Fanuc TP program (LS listing): SET_STR.LS

/PROG  SET_STR
/ATTR
OWNER		= MNEDITOR;
COMMENT		= "";
PROG_SIZE	= 228;
CREATE		= DATE 26-06-16  TIME 17:54:20;
MODIFIED	= DATE 26-06-16  TIME 17:54:20;
FILE_NAME	= SET_STR;
VERSION		= 0;
LINE_COUNT	= 2;
MEMORY_SIZE	= 592;
PROTECT		= READ_WRITE;
TCD:  STACK_SIZE	= 0,
      TASK_PRIORITY	= 50,
      TIME_SLICE	= 0,
      BUSY_LAMP_OFF	= 0,
      ABORT_REQUEST	= 0,
      PAUSE_REQUEST	= 0;
DEFAULT_GROUP	= 1,*,*,*,*;
CONTROL_CODE	= 00000000 00000000;
LOCAL_REGISTERS	= 0,0,0;
/APPL
/MN
   1:  !This program put Argument in SR ;
   2:  SR[AR[2]]=AR[1]    ;
/POS
/END
